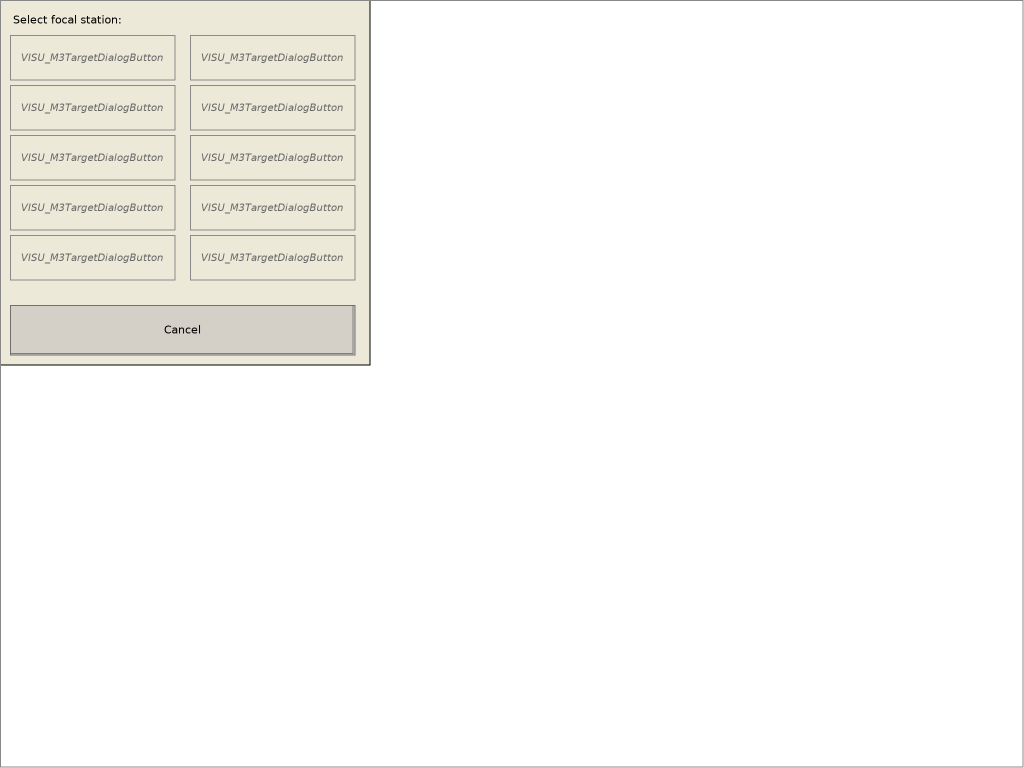
VISUALIZATION VISU_M3TargetDialog  // 1024x768
    Rectangle (0,0 370x365)
    Button (10,305 345x50), "Cancel"
        OnMouseClick: CloseDialog Dialog=VISU_M3TargetDialog, Result=Cancel, NumpadKeypadSet=True
    Label (10,5 165x30), "Select focal station:"
    Frame (10,35 165x45)
        shows VISU_M3TargetDialogButton(ref := GLOBAL.gui.m3.button_targetDialog_0)
    Frame (10,85 165x45)
        shows VISU_M3TargetDialogButton(ref := GLOBAL.gui.m3.button_targetDialog_1)
    Frame (10,135 165x45)
        shows VISU_M3TargetDialogButton(ref := GLOBAL.gui.m3.button_targetDialog_2)
    Frame (10,185 165x45)
        shows VISU_M3TargetDialogButton(ref := GLOBAL.gui.m3.button_targetDialog_3)
    Frame (10,235 165x45)
        shows VISU_M3TargetDialogButton(ref := GLOBAL.gui.m3.button_targetDialog_4)
    Frame (190,35 165x45)
        shows VISU_M3TargetDialogButton(ref := GLOBAL.gui.m3.button_targetDialog_5)
    Frame (190,85 165x45)
        shows VISU_M3TargetDialogButton(ref := GLOBAL.gui.m3.button_targetDialog_6)
    Frame (190,135 165x45)
        shows VISU_M3TargetDialogButton(ref := GLOBAL.gui.m3.button_targetDialog_7)
    Frame (190,185 165x45)
        shows VISU_M3TargetDialogButton(ref := GLOBAL.gui.m3.button_targetDialog_8)
    Frame (190,235 165x45)
        shows VISU_M3TargetDialogButton(ref := GLOBAL.gui.m3.button_targetDialog_9)
END_VISUALIZATION

(* stored: Version 1.1.0.1, ProductVersion 3.1.4019.2
   Visu VISU_M3TargetDialog: Id {4222a375-0e62-4488-88a2-1a028785d214} *)
